// Mitsubishi GX Works2 project: 28-05-2020 STL GXWorks2   PLC: FX3U/FX3UC

PROGRAM MAIN
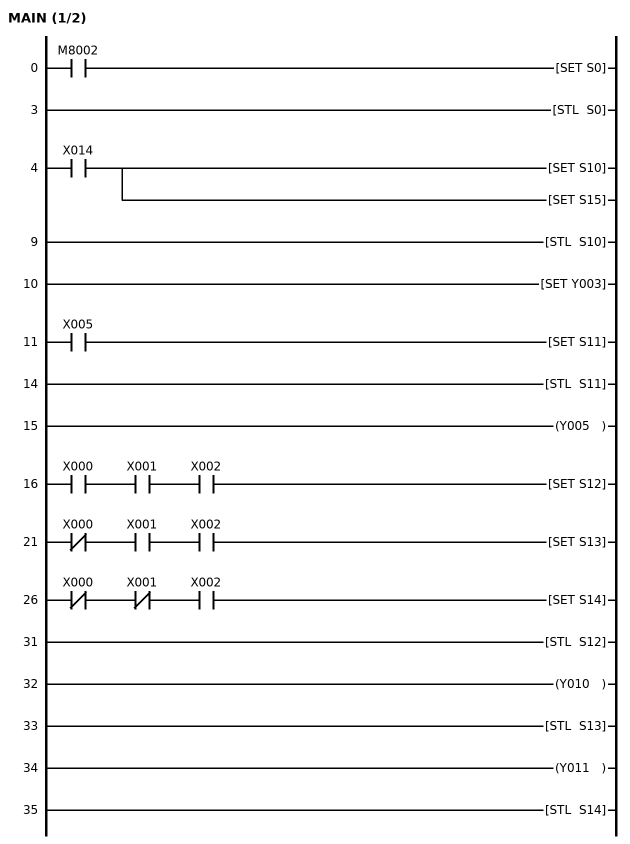
0     LD      M8002
      SET     S0
3     STL     S0
4     LD      X014
      SET     S10
      SET     S15
9     STL     S10
10    SET     Y003
11    LD      X005
      SET     S11
14    STL     S11
15    OUT     Y005
16    LD      X000
      AND     X001
      AND     X002
      SET     S12
21    LDI     X000
      AND     X001
      AND     X002
      SET     S13
26    LDI     X000
      ANI     X001
      AND     X002
      SET     S14
31    STL     S12
32    OUT     Y010
33    STL     S13
34    OUT     Y011
35    STL     S14
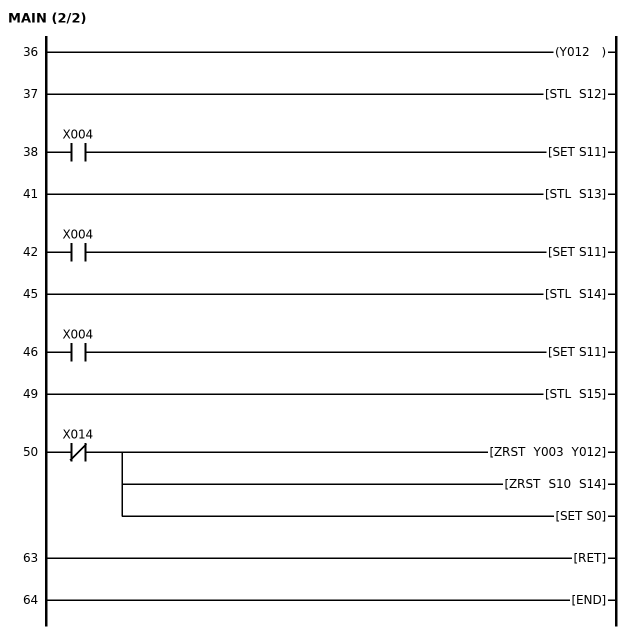
36    OUT     Y012
37    STL     S12
38    LD      X004
      SET     S11
41    STL     S13
42    LD      X004
      SET     S11
45    STL     S14
46    LD      X004
      SET     S11
49    STL     S15
50    LDI     X014
      ZRST    Y003 Y012
      ZRST    S10 S14
      SET     S0
63    RET
64    END
END_PROGRAM
